// LS Electric XG5000 project: testrung
// PLC NewPLC

PROGRAM NewProgram (task: 스캔 프로그램)

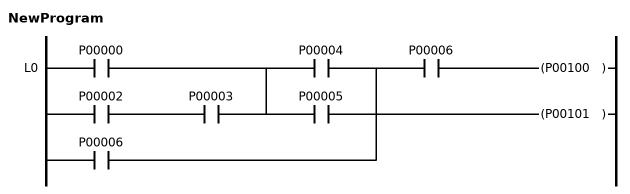
; L0
LOAD      P00000
LOAD      P00002
AND       P00003
OR LOAD
LOAD      P00004
OR        P00005
AND LOAD
OR        P00006
MPUSH
AND       P00006
OUT       P00100
MPOP
OUT       P00101